PROGRAM Axis_15_Function_Blocks
VAR
END_VAR

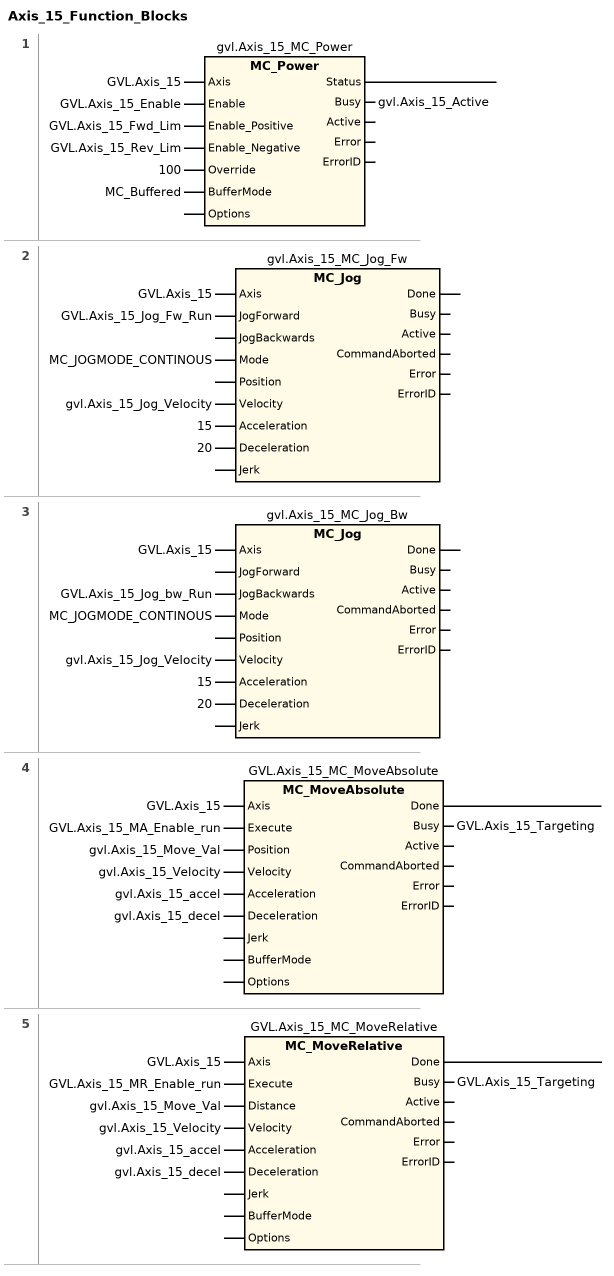
// NETWORK 1
gvl.Axis_15_MC_Power(
    Axis := GVL.Axis_15,
    Enable := GVL.Axis_15_Enable,
    Enable_Positive := GVL.Axis_15_Fwd_Lim,
    Enable_Negative := GVL.Axis_15_Rev_Lim,
    Override := 100,
    BufferMode := MC_Buffered,
    Busy => gvl.Axis_15_Active); // MC_Power

// NETWORK 2
gvl.Axis_15_MC_Jog_Fw(
    Axis := GVL.Axis_15,
    JogForward := GVL.Axis_15_Jog_Fw_Run,
    Mode := MC_JOGMODE_CONTINOUS,
    Velocity := gvl.Axis_15_Jog_Velocity,
    Acceleration := 15,
    Deceleration := 20); // MC_Jog

// NETWORK 3
gvl.Axis_15_MC_Jog_Bw(
    Axis := GVL.Axis_15,
    JogBackwards := GVL.Axis_15_Jog_bw_Run,
    Mode := MC_JOGMODE_CONTINOUS,
    Velocity := gvl.Axis_15_Jog_Velocity,
    Acceleration := 15,
    Deceleration := 20); // MC_Jog

// NETWORK 4
GVL.Axis_15_MC_MoveAbsolute(
    Axis := GVL.Axis_15,
    Execute := GVL.Axis_15_MA_Enable_run,
    Position := gvl.Axis_15_Move_Val,
    Velocity := gvl.Axis_15_Velocity,
    Acceleration := gvl.Axis_15_accel,
    Deceleration := gvl.Axis_15_decel,
    Busy => GVL.Axis_15_Targeting); // MC_MoveAbsolute

// NETWORK 5
GVL.Axis_15_MC_MoveRelative(
    Axis := GVL.Axis_15,
    Execute := GVL.Axis_15_MR_Enable_run,
    Distance := gvl.Axis_15_Move_Val,
    Velocity := gvl.Axis_15_Velocity,
    Acceleration := gvl.Axis_15_accel,
    Deceleration := gvl.Axis_15_decel,
    Busy => GVL.Axis_15_Targeting); // MC_MoveRelative

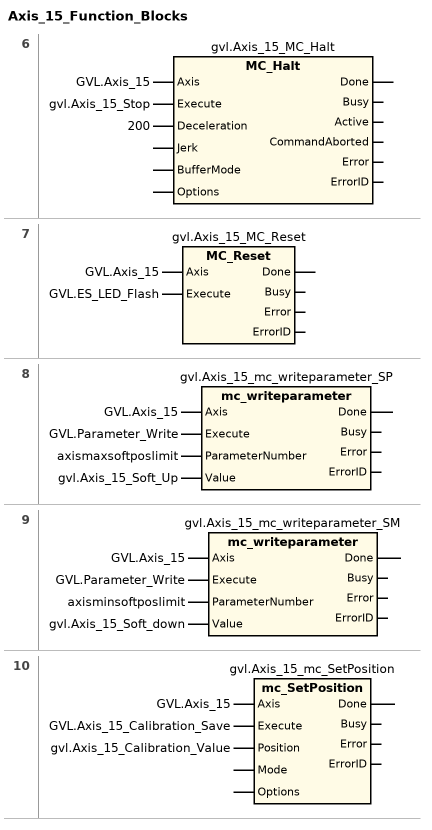
// NETWORK 6
gvl.Axis_15_MC_Halt(Axis := GVL.Axis_15, Execute := gvl.Axis_15_Stop, Deceleration := 200); // MC_Halt

// NETWORK 7
gvl.Axis_15_MC_Reset(Axis := GVL.Axis_15, Execute := GVL.ES_LED_Flash); // MC_Reset

// NETWORK 8
gvl.Axis_15_mc_writeparameter_SP(
    Axis := GVL.Axis_15,
    Execute := GVL.Parameter_Write,
    ParameterNumber := axismaxsoftposlimit,
    Value := gvl.Axis_15_Soft_Up); // mc_writeparameter

// NETWORK 9
gvl.Axis_15_mc_writeparameter_SM(
    Axis := GVL.Axis_15,
    Execute := GVL.Parameter_Write,
    ParameterNumber := axisminsoftposlimit,
    Value := gvl.Axis_15_Soft_down); // mc_writeparameter

// NETWORK 10
gvl.Axis_15_mc_SetPosition(
    Axis := GVL.Axis_15,
    Execute := GVL.Axis_15_Calibration_Save,
    Position := gvl.Axis_15_Calibration_Value); // mc_SetPosition

END_PROGRAM

(* stored: Version 1.1.0.1, ProductVersion 3.1.4022.12
   POU Axis_15_Function_Blocks: Id {5ae3e3fe-edc8-47ec-a2f4-8eec05c07737}, SpecialFunc None *)
